// STRUCT used to contain error status information.
{attribute 'enable_dynamic_creation'}
TYPE ST_ERROR :
STRUCT
	bSTATUS : BOOL; 		// Indicates if an error has occurred | TRUE = error, FALSE = no error
	nCODE 	: DINT; 		// Error code specific to the particular error.
	sSOURCE : T_MaxString; 	// Textual information describing the error.
END_STRUCT
END_TYPE

(* stored: Version 1.1.0.1, ProductVersion 3.1.4024.4
   DUT ST_ERROR: Id {770f9493-71c3-4b53-a385-4a31cd0fe4a4} *)
